{attribute addProperty BoxType "AT2050-0500-0023"}
{attribute addProperty Id "A_0090_AT2050_5501_0019_AT2050_5501AT2050_3DCFC8D064080"}
{attribute addProperty CRC "2580481503"}
{attribute addProperty SizeInBites "640"}
{attribute addProperty SizeInBytes "80"}
TYPE A_0054_AT2050_0500_0023_99CF05DF EXTENDS AT2050_9506A482 :
STRUCT
	{attribute addProperty Name "A_0090_AT2050_5501_0019_AT2050_5501"}
	A_0090_AT2050_5501_0019_AT2050_5501 : AT2050_3DCFC8D0;
END_STRUCT
END_TYPE

(* stored: Version 1.2.0.0, ProductVersion 3.1.4024.9
   DUT A_0054_AT2050_0500_0023_99CF05DF: Id {d5cb0b08-feb7-4de6-ae06-558403809906} *)
